Fanuc KAREL source: kt00296.compact.KL

PROGRAM KT00296
%STACKSIZE=65535
%PRIORITY=65535
%NOLOCKGROUP
VAR
I1 : INTEGER
H2 : ARRAY[2] OF SHORT
OUT : BOOLEAN
BEGIN
I1=2
H2[1]=3
OUT=(I1 <> H2[1])
END KT00296
